FUNCTION_BLOCK RunnerTestSuite
VAR
	TestObjRunner : ObjectRunner;
	TestMockObj : MockObj;
	ReRun : BOOL;
END_VAR

RejectInvalidInterface_Test();
IncrementObjectCountWhenAdded_Test();
IncrementInitObjCountWhenAdded_Test();
RejectAddingSameModule_Test();
RejectInitCallWithNoModules_Test();
IF ReRun THEN
	TestSuite.ReRunTests();
	ReRun := FALSE;
END_IF

METHOD IncrementInitObjCountWhenAdded_Test : BOOL
VAR_INST
	Expected : INT;
	Actual	 : INT;
END_VAR
IF TestSuite.Test(__POUNAME()).ExecuteTest() THEN
	Expected := 1;
	TestObjRunner.RegisterModule(CyclicModule := TestMockObj);
	Actual := TestObjRunner.GetInitModuleCount();
	TestSuite.Test(__POUNAME()).AssertEqual(Expected, Actual);
	TestObjRunner.DeregisterAllModules();
END_IF
END_METHOD

METHOD IncrementObjectCountWhenAdded_Test : BOOL
VAR_INST
	Expected : INT;
	Actual	 : INT;
END_VAR
IF TestSuite.Test(__POUNAME()).ExecuteTest() THEN
	Expected := 1;
	TestObjRunner.RegisterModule(CyclicModule := TestMockObj);
	Actual := TestObjRunner.GetCyclicModuleCount();
	TestSuite.Test(__POUNAME()).AssertEqual(Expected, Actual);
	TestObjRunner.DeregisterAllModules();
END_IF
END_METHOD

METHOD RejectAddingSameModule_Test : BOOL
VAR_INST
	Expected : HRESULT;
	Actual	 : HRESULT;
END_VAR
IF TestSuite.Test(__POUNAME()).ExecuteTest() THEN
	Expected := S_False;
	TestObjRunner.RegisterModule(CyclicModule := TestMockObj);
	Actual := TestObjRunner.RegisterModule(CyclicModule := TestMockObj);
	TestSuite.Test(__POUNAME()).AssertEqual(Expected, Actual);
	TestObjRunner.DeregisterAllModules();
END_IF
END_METHOD

METHOD RejectInitCallWithNoModules_Test : BOOL
VAR_INST
	Expected : HRESULT;
	Actual	 : HRESULT;
END_VAR
IF TestSuite.Test(__POUNAME()).ExecuteTest() THEN
	Expected := S_False;
	Actual := TestObjRunner.Initialise();
	TestSuite.Test(__POUNAME()).AssertEqual(Expected, Actual);
	TestObjRunner.DeregisterAllModules();
END_IF
END_METHOD

METHOD RejectInvalidInterface_Test : BOOL
VAR_INST
	Expected : HRESULT;
	Actual	 : HRESULT;
END_VAR
IF TestSuite.Test(__POUNAME()).ExecuteTest() THEN
	Expected := S_False;
	Actual := TestObjRunner.RegisterModule(CyclicModule := 16#0);
	TestSuite.Test(__POUNAME()).AssertEqual(Expected, Actual);
END_IF
END_METHOD

END_FUNCTION_BLOCK

(* stored: Version 1.1.0.1
   POU RunnerTestSuite: Id {aa66a70b-e6a1-4ee9-93b5-91581bfef23c}, SpecialFunc None
   Method IncrementInitObjCountWhenAdded_Test: Id {7128a3c1-eb86-432a-a99b-ea139722f283}
   Method IncrementObjectCountWhenAdded_Test: Id {c3a80c9e-fe7e-4a12-b8cb-4c7062482f36}
   Method RejectAddingSameModule_Test: Id {c962196c-5e81-4f84-9de9-a591b396130d}
   Method RejectInitCallWithNoModules_Test: Id {06ac3e74-0018-40e7-bbfd-7c5fde7c73e6}
   Method RejectInvalidInterface_Test: Id {1a121526-1763-4409-b8b9-2573d17baec6} *)
